Fanuc KAREL source: kt00557.KL

PROGRAM KT00557
%STACKSIZE=65535
%PRIORITY=65535
%NOLOCKGROUP
-- UNRESOLVED DECLARATIONS (source type spelling not recovered)
-- V1 : TYPE_0x0013 (type_u16=0x0013)
-- V2 : TYPE_0x0013 (type_u16=0x0013)
-- OUT : TYPE_0x0013 (type_u16=0x0013)
BEGIN
-- UNSAFE_SOURCE_IR line 8: field_offset(V1,0) = 1065353216
-- UNSAFE_SOURCE_IR line 9: field_offset(V2,4) = 1073741824
-- UNSAFE_SOURCE_IR line 10: field_offset(V1,0) = 1065353216
-- UNSAFE_SOURCE_IR line 11: field_offset(V2,4) = 1073741824
-- UNRESOLVED_PC line 12 opcodes [49 49 93 4A] marker_code=80
END KT00557
